// Mitsubishi GX Works2 project: 05.26   PLC: Q02/Q02H

PROGRAM MAIN
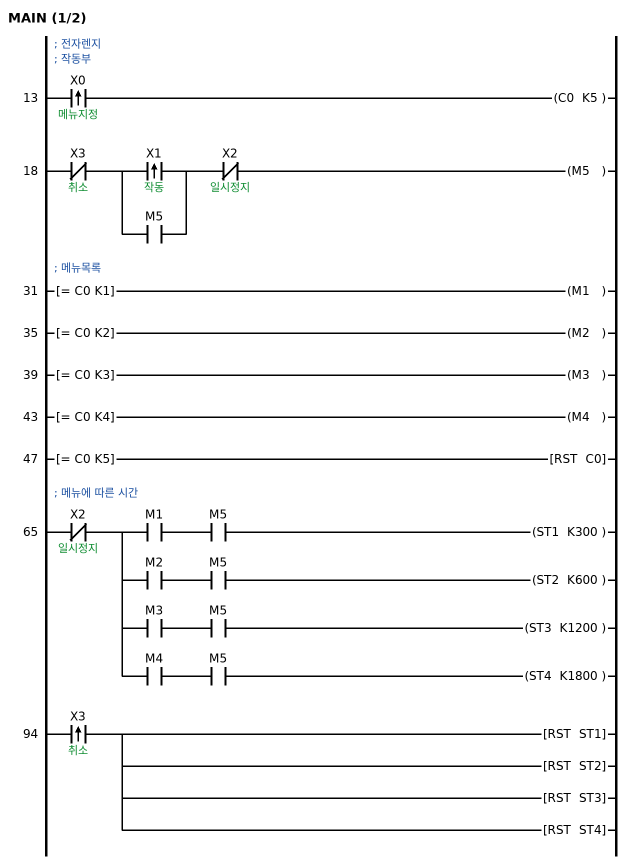
; 전자렌지
; 작동부
13    LDP     X0  ; 메뉴지정
      OUT     C0 K5
18    LDI     X3  ; 취소
      LDP     X1  ; 작동
      OR      M5
      ANB
      ANI     X2  ; 일시정지
      OUT     M5
; 메뉴목록
31    LD=     C0 K1
      OUT     M1
35    LD=     C0 K2
      OUT     M2
39    LD=     C0 K3
      OUT     M3
43    LD=     C0 K4
      OUT     M4
47    LD=     C0 K5
      RST     C0
; 메뉴에 따른 시간
65    LDI     X2  ; 일시정지
      MPS
      AND     M1
      AND     M5
      OUT     ST1 K300
      MRD
      AND     M2
      AND     M5
      OUT     ST2 K600
      MRD
      AND     M3
      AND     M5
      OUT     ST3 K1200
      MPP
      AND     M4
      AND     M5
      OUT     ST4 K1800
94    LDP     X3  ; 취소
      RST     ST1
      RST     ST2
      RST     ST3
      RST     ST4
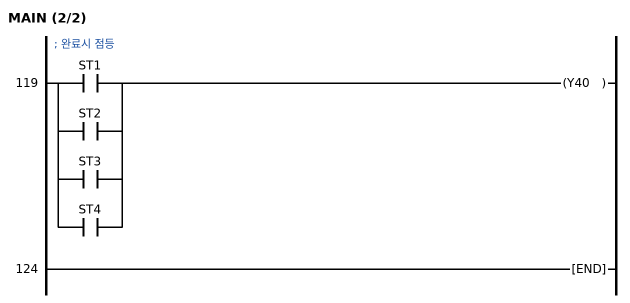
; 완료시 점등
119   LD      ST1
      OR      ST2
      OR      ST3
      OR      ST4
      OUT     Y40
124   END
END_PROGRAM
